// TIA Portal V20 export
DATA_BLOCK "HMI_Pallets"   // DB24
{ S7_Optimized_Access := 'TRUE' }
// stored: MemoryReserve 100
   VAR
      Reset_Drivers : Bool;
      Row : Int;
      Station_Row4 : Int;
      Station_Row2 : Int;
      Station_Row1 : Int;
      Run_Command_left_ROW1 : Array[1..12] of Bool;
      Run_Command_left_ROW2 : Array[1..12] of Bool;
      Run_Command_left_ROW3 : Array[1..12] of Bool;
      Run_Command_left_ROW4 : Array[1..12] of Bool;
      Run_Command_right_ROW1 : Array[1..12] of Bool;
      Run_Command_right_ROW2 : Array[1..12] of Bool;
      Run_Command_right_ROW3 : Array[1..12] of Bool;
      Run_Command_right_ROW4 : Array[1..12] of Bool;
      Run_Status_left_ROW1 : Array[1..12] of Bool;
      Run_Status_left_ROW2 : Array[1..12] of Bool;
      Run_Status_left_ROW3 : Array[1..12] of Bool;
      Run_Status_left_ROW4 : Array[1..12] of Bool;
      Run_Status_right_ROW1 : Array[1..12] of Bool;
      Run_Status_right_ROW2 : Array[1..12] of Bool;
      Run_Status_right_ROW3 : Array[1..12] of Bool;
      Run_Status_right_ROW4 : Array[1..12] of Bool;
      Number_Of_Pallet : SInt;
      Stop_Driver_Button1 : DWord;
      Stop_Driver_HMI1 : DWord;
      Stop_Driver_Button2 : DWord;
      Stop_Driver_HMI2 : DWord;
      Stop_Driver_Status : Bool;
      Drive_Error_Status : Bool;
      Command_Run_W1 : Bool;
      Command_Run_W2 : Bool;
      Command_Run_W4 : Bool;
   END_VAR
BEGIN
END_DATA_BLOCK
